(*
version 1.0	 2 dec 2007
programmer 	hugo
tested by		tobias

this function calculates the exponent to the basis 10
exp10(3) = 1000

*)
FUNCTION EXP10 : REAL
VAR_INPUT
	X : REAL;
END_VAR

EXP10 := EXP(X * 2.30258509299405);

(* revision history
hm	2. dec 2007		rev 1.0
	original version

*)

END_FUNCTION

(* stored: Version 1.1.0.1
   POU EXP10: Id {9a335cf3-a589-45b8-b8ff-4881f1499bc7}, SpecialFunc None *)
